(* CoDeSys 2.3 export: IED_BLOCK.EXP *)

(* POU IED_BLOCK, FBD *)
FUNCTION_BLOCK IED_BLOCK
VAR_INPUT
	ied_addr: 			STRING;
	ied_connect:		INT;
	gen_connect: 		INT;
	unit_id:			BYTE;
	power:				UINT;
END_VAR
VAR_OUTPUT
END_VAR
VAR
	ied_state:					INT;
	gen_state: 				INT;
	cmd: 						INT;
	ied_state_en:				BOOL;
	ied_state_done:			BOOL;
	ied_state_error: 			BOOL;
	ied_state_cts:				BOOL;
	ied_state_ctrl:				INT;
	gen_state_en:				BOOL;
	gen_state_done:			BOOL;
	gen_state_error:			BOOL;
	gen_state_cts:			BOOL;
	gen_state_ctrl:			INT;
	cmd_cts: 					BOOL;
	cmd_send:				BOOL;
	cmd_done: 				BOOL;
	ied_state_sender:		ETH_MOD_MAST;
	gen_state_sender: 		ETH_MOD_MAST;
	cmd_sender: 				ETH_MOD_MAST;
	cmd_wave: 				BLINK;
	ied_state_synch: 			IED_STATE_SYNC;
	ied_state_en_initi: 		IED_STATE_EN_INIT;
	gen_state_synch: 		GEN_STATE_SYNC;
	gen_state_en_initi: 		GEN_STATE_EN_INIT;
	cmd_synch: 				CMD_SYNC;
END_VAR
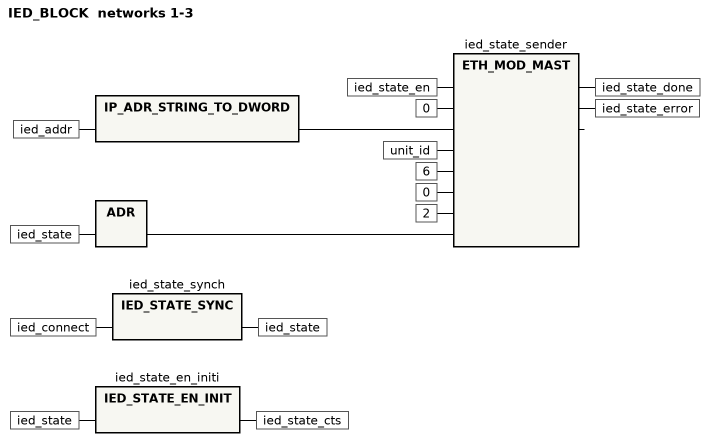
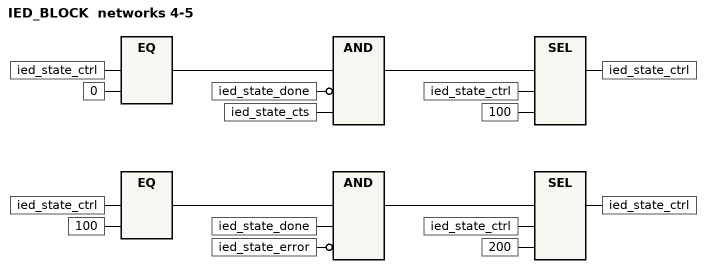
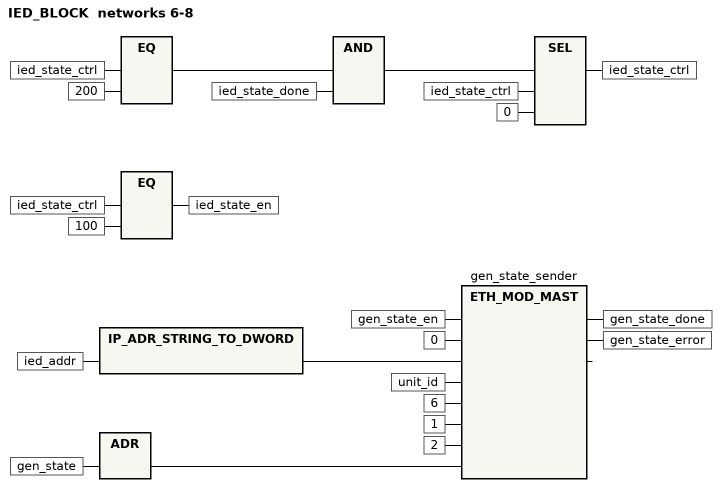
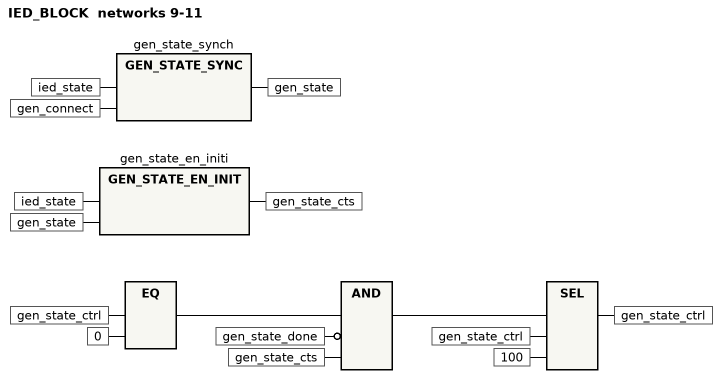
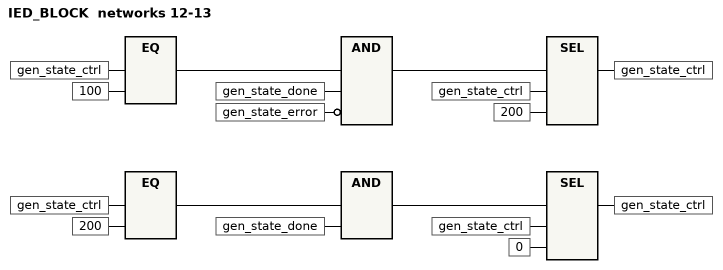
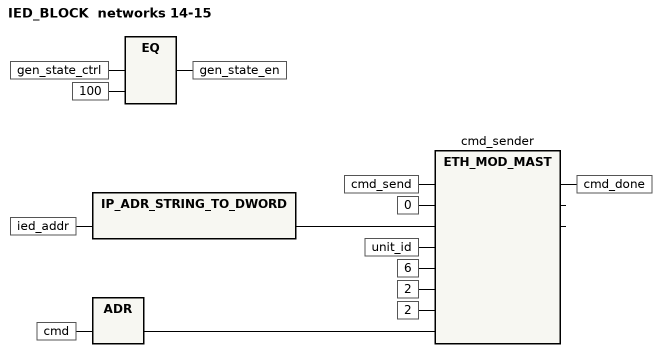
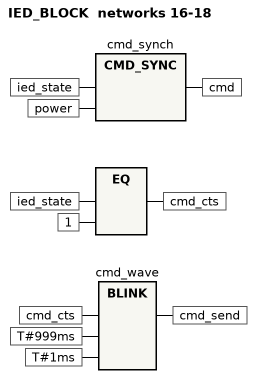
_FBD_ (* Function Block Diagram *)
NETWORK 1
	ied_state_sender:ETH_MOD_MAST(ied_state_en, 0, IP_ADR_STRING_TO_DWORD(ied_addr), unit_id, 6, 0, 2, ADR(ied_state), out 2 => ied_state_error) => ied_state_done
NETWORK 2
	ied_state_synch:IED_STATE_SYNC(ied_connect) => ied_state
NETWORK 3
	ied_state_en_initi:IED_STATE_EN_INIT(ied_state) => ied_state_cts
NETWORK 4
	SEL(AND(EQ(ied_state_ctrl, 0), NOT ied_state_done, ied_state_cts), ied_state_ctrl, 100) => ied_state_ctrl
NETWORK 5
	SEL(AND(EQ(ied_state_ctrl, 100), ied_state_done, NOT ied_state_error), ied_state_ctrl, 200) => ied_state_ctrl
NETWORK 6
	SEL(AND(EQ(ied_state_ctrl, 200), ied_state_done), ied_state_ctrl, 0) => ied_state_ctrl
NETWORK 7
	EQ(ied_state_ctrl, 100) => ied_state_en
NETWORK 8
	gen_state_sender:ETH_MOD_MAST(gen_state_en, 0, IP_ADR_STRING_TO_DWORD(ied_addr), unit_id, 6, 1, 2, ADR(gen_state), out 2 => gen_state_error) => gen_state_done
NETWORK 9
	gen_state_synch:GEN_STATE_SYNC(ied_state, gen_connect) => gen_state
NETWORK 10
	gen_state_en_initi:GEN_STATE_EN_INIT(ied_state, gen_state) => gen_state_cts
NETWORK 11
	SEL(AND(EQ(gen_state_ctrl, 0), NOT gen_state_done, gen_state_cts), gen_state_ctrl, 100) => gen_state_ctrl
NETWORK 12
	SEL(AND(EQ(gen_state_ctrl, 100), gen_state_done, NOT gen_state_error), gen_state_ctrl, 200) => gen_state_ctrl
NETWORK 13
	SEL(AND(EQ(gen_state_ctrl, 200), gen_state_done), gen_state_ctrl, 0) => gen_state_ctrl
NETWORK 14
	EQ(gen_state_ctrl, 100) => gen_state_en
NETWORK 15
	cmd_sender:ETH_MOD_MAST(cmd_send, 0, IP_ADR_STRING_TO_DWORD(ied_addr), unit_id, 6, 2, 2, ADR(cmd)) => cmd_done
NETWORK 16
	cmd_synch:CMD_SYNC(ied_state, power) => cmd
NETWORK 17
	EQ(ied_state, 1) => cmd_cts
NETWORK 18
	cmd_wave:BLINK(cmd_cts, T#999ms, T#1ms) => cmd_send
_END_FBD_
(* the same logic as Structured Text *)
(* Network 1: see the listing above *)
(* Network 2: see the listing above *)
(* Network 3: see the listing above *)
(* Network 4 *)
ied_state_ctrl := SEL((ied_state_ctrl = 0) AND NOT ied_state_done AND ied_state_cts, ied_state_ctrl, 100);
(* Network 5 *)
ied_state_ctrl := SEL((ied_state_ctrl = 100) AND ied_state_done AND NOT ied_state_error, ied_state_ctrl, 200);
(* Network 6 *)
ied_state_ctrl := SEL((ied_state_ctrl = 200) AND ied_state_done, ied_state_ctrl, 0);
(* Network 7 *)
ied_state_en := ied_state_ctrl = 100;
(* Network 8: see the listing above *)
(* Network 9: see the listing above *)
(* Network 10: see the listing above *)
(* Network 11 *)
gen_state_ctrl := SEL((gen_state_ctrl = 0) AND NOT gen_state_done AND gen_state_cts, gen_state_ctrl, 100);
(* Network 12 *)
gen_state_ctrl := SEL((gen_state_ctrl = 100) AND gen_state_done AND NOT gen_state_error, gen_state_ctrl, 200);
(* Network 13 *)
gen_state_ctrl := SEL((gen_state_ctrl = 200) AND gen_state_done, gen_state_ctrl, 0);
(* Network 14 *)
gen_state_en := gen_state_ctrl = 100;
(* Network 15: see the listing above *)
(* Network 16: see the listing above *)
(* Network 17 *)
cmd_cts := ied_state = 1;
(* Network 18: see the listing above *)
END_FUNCTION_BLOCK
